FUNCTION BYTE2st08b (* Function with empty body *)
  (* Standard: 61499-1 *)
  (* Version 1.0, 2024-02-22, franz *)
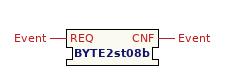
  EVENT_INPUT
    REQ;
  END_EVENT
  EVENT_OUTPUT
    CNF;
  END_EVENT
  BODY IN ST:

  END_BODY
END_FUNCTION
